// TIA Portal V17 export
// export: Created 2025-08-05T09:36:00.0345392Z, ExportSetting WithDefaults, DisplayName Totally Integrated Automation Portal, DisplayVersion V17, DisplayName TIA Portal Openness, DisplayVersion V17, DisplayName TIA Portal Version Control Interface, DisplayVersion V17, DisplayName SINAMICS Startdrive Advanced, DisplayVersion V17, DisplayName SINAMICS Startdrive G130, G150, S120, S150, SINAMICS MV, S210, DisplayVersion V17, DisplayName SINAMICS Startdrive G110M, G120, G120C, G120D, G120P, G115D, DisplayVersion V17, DisplayName STEP 7 Professional, DisplayVersion V17, DisplayName STEP 7 Safety, DisplayVersion V17, DisplayName WinCC Advanced, DisplayVersion V17
TYPE "typeGroupOvrvList"
TITLE = Overview of groups / Gruppenübersicht
// Group overview [V 01.00 | Kernel_V2] / Gruppenübersicht [V 01.00 | Kernel_V2]
// stored: IsFailsafeCompliant false
   STRUCT
      lastUsedIndex : DInt := -1;   // Letzter Benutzter Index / Last user index
      valid : Bool;   // Gültigkeit / Scope
      overflowCount : DInt;   // Gruppen Überlauf Zähler / Groups overtravel counter
      firstListedCortArea : DInt := -1;   // Index der ersten gelisteten CA / Index of first listed CA
      groups : Array[0.."MAX_CNT_GRP_OVR_ENTRIES"] of "typeGroupOvrvListEntry";   // Gruppen (CAs/CGs/FGs) / Groups (CAs/CGs/FGs)
   END_STRUCT;
END_TYPE
